(* IEC 61131-3 sources: RAG_PLC/data/result/test/026, 2 files *)

(* ---- wrapped.st ---- *)
(* =========================================================
   Generated by PLC-Eval Benchmark Wrapper
   ========================================================= *)

FUNCTION_BLOCK LLM_Wrapper_FB
VAR_INPUT
    UTC : UDINT;
    DST_ENABLE : BOOL;
    TIME_ZONE_OFFSET : INT;
END_VAR

VAR_OUTPUT
    LOCAL_TIME : UDINT;
END_VAR

VAR
    tmp : INT;
END_VAR

tmp := TIME_ZONE_OFFSET * 60;
IF DST_ENABLE THEN
    tmp := tmp + 3600;
END_IF;

IF tmp < 0 THEN
    LOCAL_TIME := UTC - _INT_TO_UDINT(ABS(tmp));
ELSE
    LOCAL_TIME := UTC + _INT_TO_UDINT(tmp);
END_IF;
END_FUNCTION_BLOCK

PROGRAM Auto_Proxy_Prg
  VAR
    instance : LLM_Wrapper_FB;
  END_VAR

  instance();
END_PROGRAM

CONFIGURATION Config0
  RESOURCE Res0 ON PLC
    TASK TaskMain(INTERVAL := T#20ms, PRIORITY := 0);
    PROGRAM Inst0 WITH TaskMain : Auto_Proxy_Prg;
  END_RESOURCE
END_CONFIGURATION

(* ---- raw_code.st ---- *)
VAR_INPUT
    UTC : UDINT;
    DST_ENABLE : BOOL;
    TIME_ZONE_OFFSET : INT;
END_VAR

VAR_OUTPUT
    LOCAL_TIME : UDINT;
END_VAR

VAR
    tmp : INT;
END_VAR

tmp := TIME_ZONE_OFFSET * 60;
IF DST_ENABLE THEN
    tmp := tmp + 3600;
END_IF;

IF tmp < 0 THEN
    LOCAL_TIME := UTC - _INT_TO_UDINT(ABS(tmp));
ELSE
    LOCAL_TIME := UTC + _INT_TO_UDINT(tmp);
END_IF;
